PROGRAM MAIN
VAR
	
END_VAR

(*
	BOUW  Alarm als berekende snelheid == 0;




*)



//PRG1_Conveyer_Operation();
//PRG2_Object_Detectie();

END_PROGRAM

(* stored: Version 1.1.0.1, ProductVersion 3.1.4024.12
   POU MAIN: Id {08eb5067-a124-4fda-bdc0-191f359724d7}, SpecialFunc None *)
